{attribute 'GeneratedUsingTerminal: EJ3202-0000-0019'}
{attribute addProperty BoxType "EJ3202-0000-0019"}
{attribute addProperty Id "RTD_Inputs_Channel_1AT %I*AI_Standard_Channel_4A3944819RTD_Inputs_Channel_2AT %I*AI_Standard_Channel_4A3944819WcStateAT %I*WcState_9091E0EB2InfoDataAT %I*InfoData_94A18F5E2"}
{attribute addProperty CRC "3364575338"}
{attribute addProperty Size "22"}
TYPE EJ3202_C88B586A EXTENDS EtcSlaveTerminalBase_947E5A46 :
STRUCT
	{attribute addProperty Name "RTD_Inputs_Channel_1"}
	RTD_Inputs_Channel_1 : AI_Standard_Channel_4A394481;
	{attribute addProperty Name "RTD_Inputs_Channel_2"}
	RTD_Inputs_Channel_2 : AI_Standard_Channel_4A394481;
	{attribute addProperty Name "WcState"}
	WcState : WcState_9091E0EB;
	{attribute addProperty Name "InfoData"}
	InfoData : InfoData_94A18F5E;
END_STRUCT
END_TYPE

(* stored: Version 1.2.0.0, ProductVersion 3.1.4024.9
   DUT EJ3202_C88B586A: Id {219b46e7-abad-4d4c-82f7-fea231c277ac} *)
